// TwinCAT 3 PLC project main
// ProgramVersion: 3.1.4024.0
// libraries:
//   Tc2_BABasic, * (Beckhoff Automation GmbH)
//   Tc2_Standard, * (Beckhoff Automation GmbH)
//   Tc2_System, * (Beckhoff Automation GmbH)
//   Tc2_Utilities, * (Beckhoff Automation GmbH)
//   Tc3_Module, * (Beckhoff Automation GmbH)
// project tree:
//   / GlobalTextList.TcGTLO, PlcTask.TcTTO, Visualization Manager.TcVMO (not stored)
//   POUs/ MAIN.TcPOU
//   VISUs/ Visu.TcVIS
// real-time tasks:
//   TASK PlcTask: cycle T#10ms, priority 20, ADS port 350

CONFIGURATION main
    RESOURCE PLC ON TwinCAT3
        TASK PlcTask(INTERVAL := T#10ms, PRIORITY := 20);
        PROGRAM MAIN WITH PlcTask : MAIN;
    END_RESOURCE
END_CONFIGURATION

// ---- POUs/MAIN.TcPOU
PROGRAM MAIN
VAR
	bAanOfUit : BOOL;
	nPot1 	: INT; //Potentiometer 1 ingestelde waarden
	nPot2 	: INT; //Potentiometer 2 huidige waarden
	bL1 	: BOOL; //Lamp
	
	DTTime : DATE_AND_TIME;
	

	
	
	
	fbTemp : FB_WeeklyTimeSwitch;
	fbTime : FB_LocalSystemTime;

	
END_VAR

//FB_WeeklyTimeSwitch -> https://infosys.beckhoff.com/english.php?content=../content/1033/tcplclibbabasic/11640109195.html&id=
//FB_LocalSystemTime -> https://infosys.beckhoff.com/english.php?content=../content/1033/tcplclib_tc2_utilities/35008651.html&id=

//Met de kamerthermostaat wordt de temperatuur in de huiskamer geregeld.
//Is de temperatuur lager dan de ingestelde waarde -1°C dan schakelt de verwarming in en als deze hoger is dan de 
//ingestelde waarde +1°C dan schakelt de verwarming uit.
//	*Potentiometer 1 bepaald de ingestelde temperatuur van 10°C tot 30°C (verschaalt).
//	*Potentiometer 2 bepaald de huidige temperatuur van -30°C tot 40°C (verschaalt).
//	*Geef de temperaturen weer via een Bar Display
//	* Een LAMP geeft aan wanneer de verwarming ingeschakeld is.

//Deze thermostaatregeling mag enkel gebeuren tijdens een bepaalde tijdsperiode, met een begin- en eindtijdstip voor iedere dag van de week.
//Gebruik hiervoor de FB_WeeklyTimeSwitch uit de TcBABasic.lib en bekijk de structure TIMESTRUCT nader voor de implementatie.
DTTime := SYSTEMTIME_TO_DT(fbTime.systemTime);

IF nPot2 < nPot1 -1 THEN
	bAanOfUit :=  TRUE;
ELSIF nPot2 > nPot1 +1 THEN
	bAanOfUit := FALSE;
END_IF

fbTemp(
	bEnable:= bAanOfUit, 
	tCurrentDateTime:= DTTime, 
	tSwitchOnTime:= TOD#11:30, 
	tSwitchOffTime:= TOD#11:55, 
	bSunday:= TRUE, 
	bMonday:= , 
	bTuesday:= , 
	bWednesday:= , 
	bThursday:= , 
	bFriday:= , 
	bSaturday:= , 
	bOutput=> bL1, 
	bEdgeOn=> , 
	bEdgeOff=> );

fbTime(
	sNetID:= , 
	bEnable:= TRUE, 
	dwCycle:=  1, 
	dwOpt:= , 
	tTimeout:= , 
	bValid=> , 
	systemTime=> , 
	tzID=> );

END_PROGRAM

// ---- VISUs/Visu.TcVIS
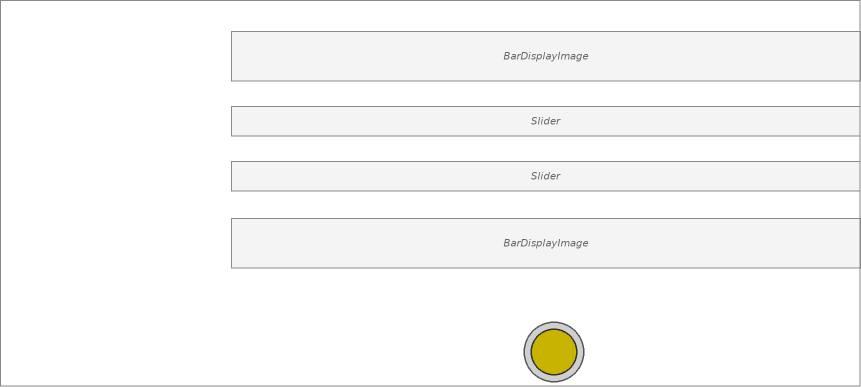
VISUALIZATION Visu  // 861x387
    Slider (231,106 629x30), variable: MAIN.nPot1, scale 10..30
    Slider (231,161 629x30), variable: MAIN.nPot2, scale -30..40
    Lamp1 (519,317 70x70), variable: MAIN.bL1, style: Lamp-Lamp1-Yellow
    BarDisplayImage (231,31 630x50), value: MAIN.nPot1, style: BarDisplayImage-Gray, scale format: %.1f, scale 10..30
    BarDisplayImage (231,218 630x50), value: MAIN.nPot2, style: BarDisplayImage-Gray, scale format: %.1f, scale -30..40
END_VISUALIZATION
